{attribute 'qualified_only'}
{attribute 'strict'}
{attribute 'to_string'}
TYPE E_Phase :
(
	L123 := 0,
	L1, 
	L2,
	L3
);
END_TYPE

(* stored: Version 1.1.0.1
   DUT E_Phase: Id {cdfbd40d-5469-0af7-01ea-c5ee3353a7ce} *)
